PROGRAM P15_RotationOperation
VAR
	rControlValue			: REAL; //rpm
	bStart_Stop				: BOOL := TRUE;
	bAlarmReset				: BOOL; //Motor Driver Alarm

	bRotationCP				: BOOL;
	nConvertedRotation_PV	: INT; //PV 0~100 rpm

	rConvertedCV			:REAL;
	(* Motor Driver *)
	bBrake_Run				: BOOL;
	(* Rotation Operation Parameter*)
	wRotaion_PV				: WORD;
	isRotationFault			: BOOL; //Motor Driver
END_VAR

VAR CONSTANT
	KL4404MaxValueP		: REAL := 16383; //0~5V, 0~3000
	//Motor Max Rotation RPM 3000rpm, Gear Ratio 20, Belt Ratio 4.5
	ConversionFactor 	: REAL :=491.49;// 491.49 ; //13106 * 20 * 4.5 / 3000
END_VAR

// Oriental Motor Driver : BLHM230K-GFS, 0~4V

_DigitalInput();

nConvertedRotation_PV := REAL_TO_INT(wRotaion_PV/(10*ConversionFactor));

// Interface with other PRGs
GVL_IO.nRotation_Converted_PV := nConvertedRotation_PV;
rControlValue := GVL_IO.rRotation_ControlValue;

//Write to Motor Driver
rConvertedCV := rControlValue * ConversionFactor; // Convert from RPM to control value

IF (GVL_IO.aController[E_aAnalogInputIO_Index.E_PV_susceptorRotation].input.targetValue > 0) OR (rConvertedCV > 0) THEN // Motor Driver RUN
	bBrake_Run := TRUE;
ELSIF (GVL_IO.aController[E_aAnalogInputIO_Index.E_PV_susceptorRotation].input.targetValue = 0) AND (rConvertedCV = 0) THEN
	bBrake_Run := FALSE;
END_IF

_DigitalOutput();

ACTION _DigitalInput:
(* Read from Power Distribution Pannel *)
bRotationCP := GVL_IO_GAS_CABINET.DI_02_RotationMotorCP;

//from Device Value
isRotationFault := NOT(GVL_IO_REACTOR_CABINET.DI_02_SusceptorRotationMotorFault);
//wRotaion_PV := UINT_TO_WORD(GVL_IO.aAnalogInputIO2[1]);
wRotaion_PV := UINT_TO_WORD(GVL_IO_REACTOR_CABINET.AI_08_R01SusceptorRotationPV);
END_ACTION

ACTION _DigitalOutput:
GVL_IO_REACTOR_CABINET.DO_05_SusceptorRotationFWD := bBrake_Run;
GVL_IO_REACTOR_CABINET.AO_09_R01_SusceptorRotationSV:=REAL_TO_INT(rConvertedCV);
 

//GVL_IO.aDigitalOutputIO[3].5 	:= bBrake_Run;
//GVL_IO.aAnalogOutputIO[28] 		:= REAL_TO_INT(rConvertedCV);
//GVL_IO.aInputState[1].11		:= isRotationFault;
END_ACTION

END_PROGRAM

(* stored: Version 1.1.0.1, ProductVersion 3.1.4024.15
   POU P15_RotationOperation: Id {7f828812-d1bb-49a4-a03d-f3e347855c39}, SpecialFunc None
   Action _DigitalInput: Id {db81d855-9855-4bd4-87ca-83883a25ba2e}
   Action _DigitalOutput: Id {b7f936ee-b5d8-4792-8a4c-a2f45c591fba} *)
